// TIA Portal V21 export
TYPE "OBJ_IODevice_IN_SICK_AFM60_Tel81_V105_Type"
   STRUCT
      ZSW2_ENC : Struct   // Encoder Status Word 2
         Bit_8 : Bool;   // Reserved
         Bit_9 : Bool;   // Control request
         Bit_10 : Bool;   // Reserved
         Bit_11 : Bool;   // Reserved
         Bit_12 : Bool;   // Encoder's Sign-of-Life
         Bit_13 : Bool;   // Encoder's Sign-of-Life
         Bit_14 : Bool;   // Encoder's Sign-of-Life
         Bit_15 : Bool;   // Encoder's Sign-of-Life
         Bit_00 : Bool;   // Reserved
         Bit_1 : Bool;   // Reserved
         Bit_2 : Bool;   // Reserved
         Bit_3 : Bool;   // Fault present
         Bit_4 : Bool;   // Reserved
         Bit_5 : Bool;   // Reserved
         Bit_6 : Bool;   // Reserved
         Bit_7 : Bool;   // Reserved
      END_STRUCT;
      G1_ZSW : Struct   // Encoder Status Word 1
         Bit_8 : Bool;   // Reserved
         Bit_9 : Bool;   // Reserved
         Bit_10 : Bool;   // Reserved
         Bit_11 : Bool;   // Requirement of error acknowledgement detected
         Bit_12 : Bool;   // Status of the preset function
         Bit_13 : Bool;   // Trasmission of absolute position value
         Bit_14 : Bool;   // Park mode activated
         Bit_15 : Bool;   // Encoder error
         Bit_00 : Bool;   // Reserved
         Bit_1 : Bool;   // Reserved
         Bit_2 : Bool;   // Reserved
         Bit_3 : Bool;   // Reserved
         Bit_4 : Bool;   // Reserved
         Bit_5 : Bool;   // Reserved
         Bit_6 : Bool;   // Reserved
         Bit_7 : Bool;   // Reserved
      END_STRUCT;
      G1_XIST1 : DInt;   // Position 1
      G1_XIST2 : DWord;   // Position 2
   END_STRUCT;
END_TYPE
